{region '#Template'}
	{attribute 'Version' := '5.0.0.0'}
	{attribute 'Tags' := '"LCID": "1031", "Text": "Universal, Control, Hysteresis"'}
	{attribute 'Tags' := '"LCID": "1033", "Text": "Universal, Control, Hysteresis"'}
	{attribute 'Using' := '"Type": "Template", "URI": "EC_ID"'}
	{attribute 'Using' := '"Type": "Template", "URI": "BA2_Param"'}
	{attribute 'Description' := '"LCID": "1031", "Text": "Hysterese"'}
	{attribute 'Description' := '"LCID": "1033", "Text": "Hysteresis"'}
{endregion}
FUNCTION_BLOCK FB_BA_Hys_03 EXTENDS FB_BA_View
VAR_INPUT
	bEn						: BOOL;
	fIn						: REAL;
END_VAR
VAR_OUTPUT
	bPresentValue			: BOOL;
	bEvent					: BOOL;	
END_VAR
VAR_INPUT CONSTANT
	On						: FB_BA_AV_Op;	
	Off						: FB_BA_AV_Op;		
	DlyOn					: FB_BA_AV_Op;	
	DlyOff					: FB_BA_AV_Op;		
	Q						: FB_BA_BV;						
END_VAR	
VAR_INPUT CONSTANT PERSISTENT
	{attribute 'parameterCategory' := 'Behaviour'}
	fOnMax					: REAL := 400.0;
	{attribute 'parameterCategory' := 'Behaviour'}
	fOffMax 				: REAL := 400.0;
END_VAR
VAR
	Swi2P					: FB_BA_Swi2P;
END_VAR

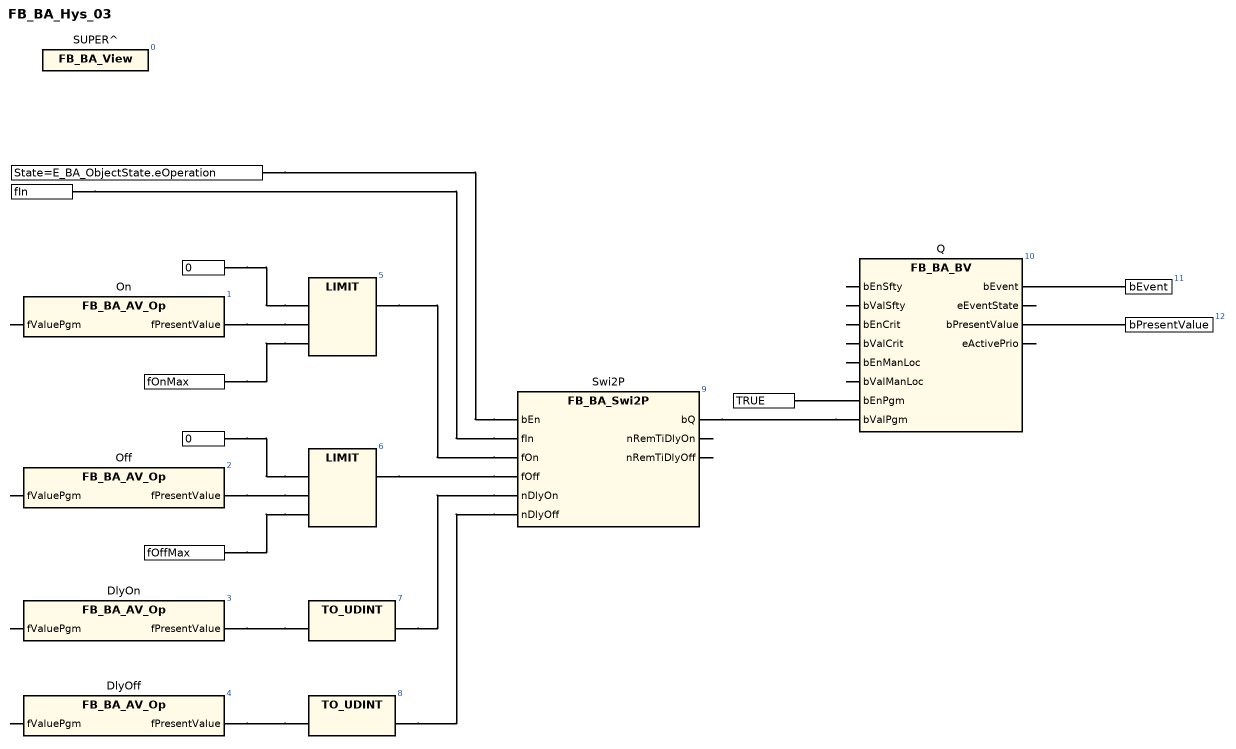
SUPER^(); // FB_BA_View
On(); // FB_BA_AV_Op
Off(); // FB_BA_AV_Op
DlyOn(); // FB_BA_AV_Op
DlyOff(); // FB_BA_AV_Op
Swi2P(
    bEn := State=E_BA_ObjectState.eOperation,
    fIn := fIn,
    fOn := LIMIT(0, On.fPresentValue, fOnMax),
    fOff := LIMIT(0, Off.fPresentValue, fOffMax),
    nDlyOn := TO_UDINT(DlyOn.fPresentValue),
    nDlyOff := TO_UDINT(DlyOff.fPresentValue)); // FB_BA_Swi2P
Q(bEnPgm := TRUE, bValPgm := Swi2P.bQ); // FB_BA_BV
bEvent := Q.bEvent;
bPresentValue := Q.bPresentValue;

METHOD FB_init : BOOL
VAR_INPUT
	bInitRetains : BOOL; // if TRUE, the retain variables are initialized (warm start / cold start)
	bInCopyCode : BOOL;  // if TRUE, the instance afterwards gets moved into the copy code (online change)
END_VAR
On.iParent							:= THIS^;
On.iLabel							:= LblFun_LimitMAX;  						 	 
On.eUnit 							:= E_BA_Unit.eTemperature_DegreesCelsius;								 
On.fValueRm							:= 18;	
On.fCOVIncrement					:= BA2_Param.fDefCOVIncrement;		

Off.iParent							:= THIS^;
Off.iLabel							:= LblFun_LimitMIN;  								 	 
Off.eUnit 							:= E_BA_Unit.eTemperature_DegreesCelsius;								 
Off.fValueRm						:= 17;			
Off.fCOVIncrement					:= BA2_Param.fDefCOVIncrement;		

DlyOn.iParent						:= THIS^;
DlyOn.iLabel						:= LblCtl_TimeDelay;
DlyOn.eUnit							:= E_BA_Unit.eTime_Seconds;
DlyOn.fValueRm						:= 30.0;

DlyOff.iParent						:= THIS^;
DlyOff.iLabel						:= LblCtl_TimeDelay;
DlyOff.eUnit						:= E_BA_Unit.eTime_Seconds;
DlyOff.fValueRm						:= 30.0;

Q.iParent							:= THIS^;
Q.iLabel							:= LblFun_SwitchingCommand;  ;	
Q.sActiveText 						:= txtEvent_Triggered;
Q.sInactiveText 					:= txtEvent_Normal;
Q.bEnManualRm						:= FALSE;	//	Priority  8	
Q.bValManualRm						:= FALSE;	//	Priority  8
Q.nEventClassID						:= EC_ID.NC30;
Q.stTimeDelay.nToNormal				:= 0;
Q.stTimeDelay.nToAbnormal			:= 0;
Q.bAlarmValue						:= TRUE;
Q.aEventTransitionText[1]			:= txtEvent_Triggered;
Q.aEventTransitionText[2]			:= txtEvent_Error;
Q.aEventTransitionText[3]			:= txtEvent_Normal;
Q.bEventDetectionEnable				:= FALSE;
Q.eEnPlantLock						:= E_BA_LockPriority.eNoLock;
END_METHOD

END_FUNCTION_BLOCK

(* stored: Version 1.1.0.1, ProductVersion 3.1.4024.12
   POU FB_BA_Hys_03: Id {ca16df4e-cb7c-41db-9e09-6bf8b3969598}, SpecialFunc None
   Method FB_init: Id {07b3ac35-d451-4e18-91b8-db36287817be} *)
